KUKA KRL program: p01drop_newold.src, p01drop_newold.dat

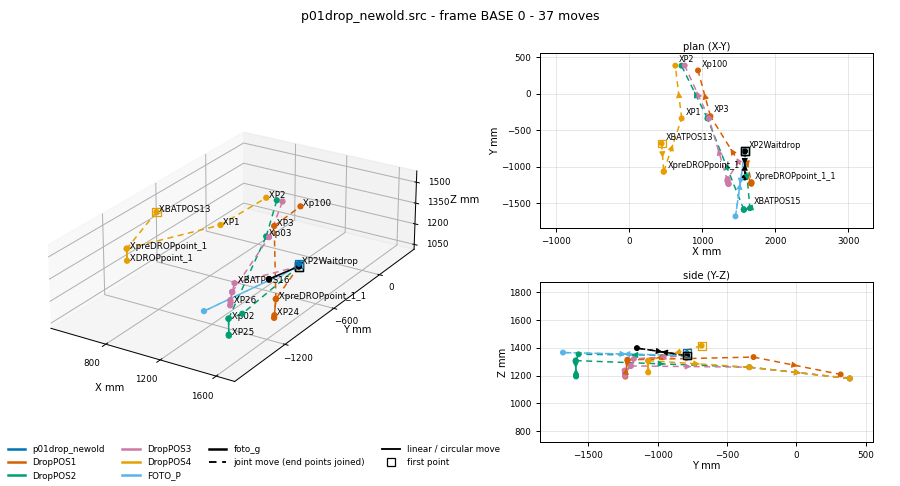
[picture p0: tool path of p01drop_newold.src in frame BASE 0, 37 of 40 moves have a stored position in this frame; points joined in program order, loops and branches not executed]
--- p01drop_newold.src ---
&ACCESS RVO1
&COMMENT Drop Part
&PARAM EDITMASK = *
&PARAM TEMPLATE = C:\KRC\Roboter\Template\vorgabe
&PARAM DISKPATH = KRC:\R1\Program\Sub Programs
DEF p01drop_newold( )
;FOLD INI
  ;FOLD BASISTECH INI

    GLOBAL INTERRUPT DECL 3 WHEN $STOPMESS==TRUE DO IR_STOPM ( )
    INTERRUPT ON 3
    BAS (#INITMOV,0 )
  ;ENDFOLD (BASISTECH INI)
;ENDFOLD (INI)
;================================================
; MODEL    : XXXX
; IE GROUP : XX
; STATION  : XXX
; ROBOT    : RX
; FUNCTION : Drop Part in StXX
;================================================
$TIMER[7]=0
$TIMER_STOP[7]=FALSE

waitarea:
QR_NOK=FALSE

;Wait For Area / Goto Safety / Return To Home
;FOLD PTP P2Waitdrop Vel=100 % PDAT2 Tool[8] Base[0];%{PE}%R 8.3.48,%MKUKATPBASIS,%CMOVE,%VPTP,%P 1:PTP, 2:P2Waitdrop, 3:, 5:100, 7:PDAT2
$BWDSTART=FALSE
PDAT_ACT=PPDAT2
FDAT_ACT=FP2Waitdrop
BAS(#PTP_PARAMS,100)
PTP XP2Waitdrop
;ENDFOLD

WAIT FOR ($IN[54]==TRUE) OR ($IN[1]==TRUE)

IF $in[54]==TRUE THEN
   bomberos_2 ( )               ; PICK In Station XX
ENDIF


;IF FALSE THEN

;Para de contar TC hasta que recibe typinfo para dejar (paleta indexada, tipo...)
$TIMER_STOP[7]=TRUE

;FOLD TYPE INFO

O_TYPE_REQ=FALSE
WAIT FOR I_TYPE_INFO==0
O_TYPE_REQ=TRUE
WAIT FOR ((I_TYPE_INFO>100) AND (I_TYPE_INFO<201) or ($IN[54]==TRUE))
IF $in[54]==TRUE THEN
   bomberos_2 ( )               ; PICK In Station XX
ENDIF
O_TYPE_INFO=I_TYPE_INFO

;ENDFOLD

;ENDIF

$TIMER_STOP[7]=FALSE

SWITCH i_TYPE_INFO ;coldplate grande o peq

CASE 111
$TIMER_STOP[7]=TRUE
INDICE_DROP=1

   O_TYPE_REQ=FALSE
;FOLD Fordtech.Area_Req Area Request: 3, Safety Position: 0, Return To Home: 0 ;%{PE}
Area_Req (3,0,0)
IF I_RETHP AND (0 <> 0) AND ($IN_HOME == TRUE) THEN
  GOTO PEXIT
ENDIF
;ENDFOLD
   $TIMER_STOP[7]=FALSE
   DropPOS1() ;POSICION 1 COLDPLATE GRANDE


CASE 112
$TIMER_STOP[7]=TRUE
INDICE_DROP=2

   O_TYPE_REQ=FALSE
;FOLD Fordtech.Area_Req Area Request: 3, Safety Position: 0, Return To Home: 0 ;%{PE}
Area_Req (3,0,0)
IF I_RETHP AND (0 <> 0) AND ($IN_HOME == TRUE) THEN
  GOTO PEXIT
ENDIF
;ENDFOLD
   $TIMER_STOP[7]=FALSE
   DropPOS2() ;POSICION 2 COLDPLATE GRANDE

CASE 113
$TIMER_STOP[7]=TRUE
INDICE_DROP=3

   O_TYPE_REQ=FALSE
;FOLD Fordtech.Area_Req Area Request: 3, Safety Position: 0, Return To Home: 0 ;%{PE}
Area_Req (3,0,0)
IF I_RETHP AND (0 <> 0) AND ($IN_HOME == TRUE) THEN
  GOTO PEXIT
ENDIF
;ENDFOLD
   $TIMER_STOP[7]=FALSE
   DropPOS3() ;POSICION 3 COLDPLATE GRANDE

CASE 150
bomberos_2 ()



CASE 121
$TIMER_STOP[7]=TRUE
INDICE_DROP=4

   O_TYPE_REQ=FALSE
;FOLD Fordtech.Area_Req Area Request: 3, Safety Position: 0, Return To Home: 0 ;%{PE}
Area_Req (3,0,0)
IF I_RETHP AND (0 <> 0) AND ($IN_HOME == TRUE) THEN
  GOTO PEXIT
ENDIF
;ENDFOLD
   $TIMER_STOP[7]=FALSE
   DropPOS1();POSICION 1 COLDPLATE PEQUEÑO

CASE 200
$TIMER_STOP[7]=TRUE
INDICE_DROP=4

   O_TYPE_REQ=FALSE
   P01DROP2_2();POSICION 1 COLDPLATE PEQUEÑO

DEFAULT

WAIT FOR FALSE

ENDSWITCH

;fold QR NOK
IF (QR_NOK==TRUE) THEN

GOTO waitarea
ENDIF

;ENDFOLD


;FOLD PROVISIONAL PARA PRUEBAS
IF M2_TYPE_INFO<13 THEN
M2_TYPE_INFO=M2_TYPE_INFO+1
ENDIF

;ENDFOLD

PEXIT:

;FOLD Guarda_TC Dejada

;Guarda TC dejada
$TIMER_STOP[7]=TRUE
TC_DROP[INDICE_DROP]=$TIMER[7]

IF (INDICE_DROP < 4) THEN ;CUANDO DEJA ARRAYS EN COLD PLATES GRANDES
   IF (INDICE_RACK == 1)THEN
      TC_CP_BIG[INDICE_DROP]=TC_DROP[INDICE_DROP]+TC_PICK_RACK1[INDICE_PICK]
   ELSE
      TC_CP_BIG[INDICE_DROP]=TC_DROP[INDICE_DROP]+TC_PICK_RACK2[INDICE_PICK]
   ENDIF
   IF (INDICE_DROP == 3) THEN ;Cuando rellena el tercer colplate acumula en array de CP big
      TC_ARRAY_CPB[INDICE_ARRAYS_CPB]=TC_CP_BIG[1]+TC_CP_BIG[2]+TC_CP_BIG[3]
      INDICE_ARRAYS_CPB=INDICE_ARRAYS_CPB+1
      IF (INDICE_ARRAYS_CPB > 18) THEN
         INDICE_ARRAYS_CPB=1
         ;Actualiza el tiempo de ciclo medio por bateria
         ;Toma el tiempo de ciclo medio por batería como la media de procesar 2 racks
         ;64 arrays y 4 cartones, eso vienen a ser unas 7 baterías y me sobra 1 array
         TC_MEDIO_CARTONES=((((TC_CARTON[1]+TC_CARTON[2]+TC_CARTON[3]+TC_CARTON[4])/1000)*63)/64)
         TC_MEDIO_BATERIA=((TC_ARRAY_CPB[1]+TC_ARRAY_CPB[2]+TC_ARRAY_CPB[3]+TC_ARRAY_CPB[4]+TC_ARRAY_CPB[5]+TC_ARRAY_CPB[6]+TC_ARRAY_CPB[7]+TC_ARRAY_CPB[8]+TC_ARRAY_CPB[9]+TC_ARRAY_CPB[10]+TC_ARRAY_CPB[11]+TC_ARRAY_CPB[12]+TC_ARRAY_CPB[13]+TC_ARRAY_CPB[14]+TC_ARRAY_CPB[15]+TC_ARRAY_CPB[16]+TC_ARRAY_CPB[17]+TC_ARRAY_CPB[18]+TC_CP_SMALL[1]+TC_CP_SMALL[2]+TC_CP_SMALL[3]+TC_CP_SMALL[4]+TC_CP_SMALL[5]+TC_CP_SMALL[6]+TC_CP_SMALL[7]+TC_CP_SMALL[8]+TC_CP_SMALL[9])/1000)
         TC_MEDIO_BATERIA=((TC_MEDIO_BATERIA+TC_MEDIO_CARTONES)/9)
      ENDIF
   ENDIF
      ENDIF

IF (INDICE_DROP == 4) THEN ;CUANDO DEJA ARRAYS EN COLD PLATE PEQUEÑOS
   IF (INDICE_RACK == 1)THEN
      TC_CP_SMALL[INDICE_ARRAYS_CPS]=TC_DROP[4]+TC_PICK_RACK1[INDICE_PICK]
   ELSE
      TC_CP_SMALL[INDICE_ARRAYS_CPS]=TC_DROP[4]+TC_PICK_RACK2[INDICE_PICK]
   ENDIF
   INDICE_ARRAYS_CPS=INDICE_ARRAYS_CPS+1
   IF (INDICE_ARRAYS_CPS > 9) THEN
      INDICE_ARRAYS_CPS=1
   ENDIF
ENDIF

;ENDFOLD

END
DEF       DropPOS1()



;FOLD PTP P11 CONT Vel=100 % PDAT29 Tool[8] Base[0];%{PE}%R 8.3.48,%MKUKATPBASIS,%CMOVE,%VPTP,%P 1:PTP, 2:P11, 3:C_DIS, 5:100, 7:PDAT29
$BWDSTART=FALSE
PDAT_ACT=PPDAT29
FDAT_ACT=FP11
BAS(#PTP_PARAMS,100)
PTP XP11 C_DIS
;ENDFOLD

;Wait For Area / Goto Safety / Return To Home

;FOLD PTP preDROPpoint_1_1 CONT Vel=100 % PDAT9 Tool[8] Base[0];%{PE}%R 8.3.48,%MKUKATPBASIS,%CMOVE,%VPTP,%P 1:PTP, 2:preDROPpoint_1_1, 3:C_DIS, 5:100, 7:PDAT9
$BWDSTART=FALSE
PDAT_ACT=PPDAT9
FDAT_ACT=FpreDROPpoint_1_1
BAS(#PTP_PARAMS,100)
PTP XpreDROPpoint_1_1 C_DIS
;ENDFOLD

;FOLD LIN P24 CONT Vel=2 m/s CPDAT10 Tool[8] Base[0];%{PE}%R 8.3.48,%MKUKATPBASIS,%CMOVE,%VLIN,%P 1:LIN, 2:P24, 3:C_DIS C_DIS, 5:2, 7:CPDAT10
$BWDSTART=FALSE
LDAT_ACT=LCPDAT10
FDAT_ACT=FP24
BAS(#CP_PARAMS,2)
LIN XP24 C_DIS C_DIS
;ENDFOLD
;FOLD LIN DROPpoint_1_1 Vel=0.02 m/s L Tool[8] Base[0];%{PE}%R 8.3.48,%MKUKATPBASIS,%CMOVE,%VLIN,%P 1:LIN, 2:DROPpoint_1_1, 3:, 5:0.02, 7:L
$BWDSTART=FALSE
LDAT_ACT=LL
FDAT_ACT=FDROPpoint_1_1
BAS(#CP_PARAMS,0.02)
LIN XDROPpoint_1_1
;ENDFOLD


;chequeo finales de carrera pieza ON
;FOLD WAIT FOR ( IN 257 'F carrera superior S202' );%{PE}%R 8.3.48,%MKUKATPBASIS,%CEXT_WAIT_FOR,%VEXT_WAIT_FOR,%P 2:, 4:, 5:$IN, 6:257, 7:F carrera superior S202, 9:
WAIT FOR  ( $IN[257] )
;ENDFOLD
;FOLD WAIT FOR ( IN 258 'F carrera superior S201' );%{PE}%R 8.3.48,%MKUKATPBASIS,%CEXT_WAIT_FOR,%VEXT_WAIT_FOR,%P 2:, 4:, 5:$IN, 6:258, 7:F carrera superior S201, 9:
WAIT FOR  ( $IN[258] )
;ENDFOLD

;abrir gara
cil_bat_reposo()

;chequeo sensores pieza OFF
;FOLD WAIT FOR NOT ( IN 243 'Partcheck array LH S501' );%{PE}%R 8.3.48,%MKUKATPBASIS,%CEXT_WAIT_FOR,%VEXT_WAIT_FOR,%P 2:NOT, 4:, 5:$IN, 6:243, 7:Partcheck array LH S501, 9:
WAIT FOR  NOT ( $IN[243] )
;ENDFOLD
;FOLD WAIT FOR NOT ( IN 244 'Partcheck array RH S502' );%{PE}%R 8.3.48,%MKUKATPBASIS,%CEXT_WAIT_FOR,%VEXT_WAIT_FOR,%P 2:NOT, 4:, 5:$IN, 6:244, 7:Partcheck array RH S502, 9:
WAIT FOR  NOT ( $IN[244] )
;ENDFOLD

;FOLD PTP preDROPpoint_1_1 CONT Vel=70 % PDAT20 Tool[8] Base[0];%{PE}%R 8.3.48,%MKUKATPBASIS,%CMOVE,%VPTP,%P 1:PTP, 2:preDROPpoint_1_1, 3:C_DIS, 5:70, 7:PDAT20
$BWDSTART=FALSE
PDAT_ACT=PPDAT20
FDAT_ACT=FpreDROPpoint_1_1
BAS(#PTP_PARAMS,70)
PTP XpreDROPpoint_1_1 C_DIS
;ENDFOLD

;chequeo finales de carrera pieza OFF
;FOLD WAIT FOR NOT ( IN 257 'F carrera superior S202' );%{PE}%R 8.3.48,%MKUKATPBASIS,%CEXT_WAIT_FOR,%VEXT_WAIT_FOR,%P 2:NOT, 4:, 5:$IN, 6:257, 7:F carrera superior S202, 9:
WAIT FOR  NOT ( $IN[257] )
;ENDFOLD
;FOLD WAIT FOR NOT ( IN 258 'F carrera superior S201' );%{PE}%R 8.3.48,%MKUKATPBASIS,%CEXT_WAIT_FOR,%VEXT_WAIT_FOR,%P 2:NOT, 4:, 5:$IN, 6:258, 7:F carrera superior S201, 9:
WAIT FOR  NOT ( $IN[258] )
;ENDFOLD

;FOLD SYN OUT 43 'Job Ready 3' State=TRUE at START Delay=0 ms;%{PE}%R 8.3.48,%MKUKATPBASIS,%COUT,%VSYNOUT,%P 2:43, 3:Job Ready 3, 5:TRUE, 7:0, 9:0, 12:0
TRIGGER WHEN DISTANCE=0 DELAY=0 DO $OUT[43]=TRUE
;ENDFOLD



;FOLD PTP P3 CONT Vel=100 % PDAT9 Tool[5] Base[0];%{PE}%R 8.3.48,%MKUKATPBASIS,%CMOVE,%VPTP,%P 1:PTP, 2:P3, 3:C_DIS, 5:100, 7:PDAT9
$BWDSTART=FALSE
PDAT_ACT=PPDAT9
FDAT_ACT=FP3
BAS(#PTP_PARAMS,100)
PTP XP3 C_DIS
;ENDFOLD

;Release Area 1
;FOLD SYN OUT 19 'Area Release 3' State=TRUE at START Delay=0 ms;%{PE}%R 8.3.48,%MKUKATPBASIS,%COUT,%VSYNOUT,%P 2:19, 3:Area Release 3, 5:TRUE, 7:0, 9:0, 12:0
TRIGGER WHEN DISTANCE=0 DELAY=0 DO $OUT[19]=TRUE
;ENDFOLD

;FOLD PTP p100 CONT Vel=100 % PDAT23 Tool[5] Base[0];%{PE}%R 8.3.48,%MKUKATPBASIS,%CMOVE,%VPTP,%P 1:PTP, 2:p100, 3:C_DIS, 5:100, 7:PDAT23
$BWDSTART=FALSE
PDAT_ACT=PPDAT23
FDAT_ACT=Fp100
BAS(#PTP_PARAMS,100)
PTP Xp100 C_DIS
;ENDFOLD


;FOLD PTP HOME Vel=100 % DEFAULT;%{PE}%R 8.3.48,%MKUKATPBASIS,%CMOVE,%VPTP,%P 1:PTP, 2:HOME, 3:, 5:100, 7:DEFAULT
$BWDSTART=FALSE
PDAT_ACT=PDEFAULT
FDAT_ACT=FHOME
BAS(#PTP_PARAMS,100)
$H_POS=XHOME
PTP XHOME
;ENDFOLD
;Jump Adress
PEXIT:



END

DEF       DropPOS2()


;FOLD PTP P12 CONT Vel=100 % PDAT30 Tool[8] Base[0];%{PE}%R 8.3.48,%MKUKATPBASIS,%CMOVE,%VPTP,%P 1:PTP, 2:P12, 3:C_DIS, 5:100, 7:PDAT30
$BWDSTART=FALSE
PDAT_ACT=PPDAT30
FDAT_ACT=FP12
BAS(#PTP_PARAMS,100)
PTP XP12 C_DIS
;ENDFOLD

;FOLD PTP BATPOS15 CONT Vel=100 % PDAT11 Tool[8] Base[0];%{PE}%R 8.3.48,%MKUKATPBASIS,%CMOVE,%VPTP,%P 1:PTP, 2:BATPOS15, 3:C_DIS, 5:100, 7:PDAT11
$BWDSTART=FALSE
PDAT_ACT=PPDAT11
FDAT_ACT=FBATPOS15
BAS(#PTP_PARAMS,100)
PTP XBATPOS15 C_DIS
;ENDFOLD
;Wait For Area / Goto Safety / Return To Home
;predrop pos
;FOLD PTP p02 CONT Vel=100 % PDAT12 Tool[8] Base[0];%{PE}%R 8.3.48,%MKUKATPBASIS,%CMOVE,%VPTP,%P 1:PTP, 2:p02, 3:C_DIS, 5:100, 7:PDAT12
$BWDSTART=FALSE
PDAT_ACT=PPDAT12
FDAT_ACT=Fp02
BAS(#PTP_PARAMS,100)
PTP Xp02 C_DIS
;ENDFOLD
;FOLD LIN P25 CONT Vel=2 m/s CPDAT11 Tool[8] Base[0];%{PE}%R 8.3.48,%MKUKATPBASIS,%CMOVE,%VLIN,%P 1:LIN, 2:P25, 3:C_DIS C_DIS, 5:2, 7:CPDAT11
$BWDSTART=FALSE
LDAT_ACT=LCPDAT11
FDAT_ACT=FP25
BAS(#CP_PARAMS,2)
LIN XP25 C_DIS C_DIS
;ENDFOLD
;drop pos
;FOLD LIN p01 Vel=0.02 m/s L Tool[8] Base[0];%{PE}%R 8.3.48,%MKUKATPBASIS,%CMOVE,%VLIN,%P 1:LIN, 2:p01, 3:, 5:0.02, 7:L
$BWDSTART=FALSE
LDAT_ACT=LL
FDAT_ACT=Fp01
BAS(#CP_PARAMS,0.02)
LIN Xp01
;ENDFOLD

;chequeo finales de carrera pieza ON
;FOLD WAIT FOR ( IN 257 'F carrera superior S202' );%{PE}%R 8.3.48,%MKUKATPBASIS,%CEXT_WAIT_FOR,%VEXT_WAIT_FOR,%P 2:, 4:, 5:$IN, 6:257, 7:F carrera superior S202, 9:
WAIT FOR  ( $IN[257] )
;ENDFOLD
;FOLD WAIT FOR ( IN 258 'F carrera superior S201' );%{PE}%R 8.3.48,%MKUKATPBASIS,%CEXT_WAIT_FOR,%VEXT_WAIT_FOR,%P 2:, 4:, 5:$IN, 6:258, 7:F carrera superior S201, 9:
WAIT FOR  ( $IN[258] )
;ENDFOLD

;abrir gara
cil_bat_reposo()

;chequeo sensores pieza OFF
;FOLD WAIT FOR NOT ( IN 243 'Partcheck array LH S501' );%{PE}%R 8.3.48,%MKUKATPBASIS,%CEXT_WAIT_FOR,%VEXT_WAIT_FOR,%P 2:NOT, 4:, 5:$IN, 6:243, 7:Partcheck array LH S501, 9:
WAIT FOR  NOT ( $IN[243] )
;ENDFOLD
;FOLD WAIT FOR NOT ( IN 244 'Partcheck array RH S502' );%{PE}%R 8.3.48,%MKUKATPBASIS,%CEXT_WAIT_FOR,%VEXT_WAIT_FOR,%P 2:NOT, 4:, 5:$IN, 6:244, 7:Partcheck array RH S502, 9:
WAIT FOR  NOT ( $IN[244] )
;ENDFOLD

;FOLD PTP p02 CONT Vel=70 % PDAT21 Tool[8] Base[0];%{PE}%R 8.3.48,%MKUKATPBASIS,%CMOVE,%VPTP,%P 1:PTP, 2:p02, 3:C_DIS, 5:70, 7:PDAT21
$BWDSTART=FALSE
PDAT_ACT=PPDAT21
FDAT_ACT=Fp02
BAS(#PTP_PARAMS,70)
PTP Xp02 C_DIS
;ENDFOLD


;chequeo finales de carrera pieza OFF
;FOLD WAIT FOR NOT ( IN 257 'F carrera superior S202' );%{PE}%R 8.3.48,%MKUKATPBASIS,%CEXT_WAIT_FOR,%VEXT_WAIT_FOR,%P 2:NOT, 4:, 5:$IN, 6:257, 7:F carrera superior S202, 9:
WAIT FOR  NOT ( $IN[257] )
;ENDFOLD
;FOLD WAIT FOR NOT ( IN 258 'F carrera superior S201' );%{PE}%R 8.3.48,%MKUKATPBASIS,%CEXT_WAIT_FOR,%VEXT_WAIT_FOR,%P 2:NOT, 4:, 5:$IN, 6:258, 7:F carrera superior S201, 9:
WAIT FOR  NOT ( $IN[258] )
;ENDFOLD

;FOLD SYN OUT 43 'Job Ready 3' State=TRUE at START Delay=0 ms;%{PE}%R 8.3.48,%MKUKATPBASIS,%COUT,%VSYNOUT,%P 2:43, 3:Job Ready 3, 5:TRUE, 7:0, 9:0, 12:0
TRIGGER WHEN DISTANCE=0 DELAY=0 DO $OUT[43]=TRUE
;ENDFOLD

;FOLD PTP p03 CONT Vel=100 % PDAT13 Tool[5] Base[0];%{PE}%R 8.3.48,%MKUKATPBASIS,%CMOVE,%VPTP,%P 1:PTP, 2:p03, 3:C_DIS, 5:100, 7:PDAT13
$BWDSTART=FALSE
PDAT_ACT=PPDAT13
FDAT_ACT=Fp03
BAS(#PTP_PARAMS,100)
PTP Xp03 C_DIS
;ENDFOLD

;Release Area 1
;FOLD SYN OUT 19 'Area Release 3' State=TRUE at START Delay=0 ms;%{PE}%R 8.3.48,%MKUKATPBASIS,%COUT,%VSYNOUT,%P 2:19, 3:Area Release 3, 5:TRUE, 7:0, 9:0, 12:0
TRIGGER WHEN DISTANCE=0 DELAY=0 DO $OUT[19]=TRUE
;ENDFOLD


;FOLD PTP p04 CONT Vel=100 % PDAT14 Tool[5] Base[0];%{PE}%R 8.3.48,%MKUKATPBASIS,%CMOVE,%VPTP,%P 1:PTP, 2:p04, 3:C_DIS, 5:100, 7:PDAT14
$BWDSTART=FALSE
PDAT_ACT=PPDAT14
FDAT_ACT=Fp04
BAS(#PTP_PARAMS,100)
PTP Xp04 C_DIS
;ENDFOLD

;FOLD PTP HOME Vel=100 % DEFAULT;%{PE}%R 8.3.48,%MKUKATPBASIS,%CMOVE,%VPTP,%P 1:PTP, 2:HOME, 3:, 5:100, 7:DEFAULT
$BWDSTART=FALSE
PDAT_ACT=PDEFAULT
FDAT_ACT=FHOME
BAS(#PTP_PARAMS,100)
$H_POS=XHOME
PTP XHOME
;ENDFOLD
;Jump Adress
PEXIT:

END
DEF       DropPOS3()


;FOLD PTP P13 CONT Vel=100 % PDAT31 Tool[8] Base[0];%{PE}%R 8.3.48,%MKUKATPBASIS,%CMOVE,%VPTP,%P 1:PTP, 2:P13, 3:C_DIS, 5:100, 7:PDAT31
$BWDSTART=FALSE
PDAT_ACT=PPDAT31
FDAT_ACT=FP13
BAS(#PTP_PARAMS,100)
PTP XP13 C_DIS
;ENDFOLD

;FOLD PTP BATPOS16 CONT Vel=100 % PDAT17 Tool[8] Base[0];%{PE}%R 8.3.48,%MKUKATPBASIS,%CMOVE,%VPTP,%P 1:PTP, 2:BATPOS16, 3:C_DIS, 5:100, 7:PDAT17
$BWDSTART=FALSE
PDAT_ACT=PPDAT17
FDAT_ACT=FBATPOS16
BAS(#PTP_PARAMS,100)
PTP XBATPOS16 C_DIS
;ENDFOLD
;Wait For Area / Goto Safety / Return To Home
;predroppos
;FOLD PTP p06 CONT Vel=100 % PDAT16 Tool[8] Base[0];%{PE}%R 8.3.48,%MKUKATPBASIS,%CMOVE,%VPTP,%P 1:PTP, 2:p06, 3:C_DIS, 5:100, 7:PDAT16
$BWDSTART=FALSE
PDAT_ACT=PPDAT16
FDAT_ACT=Fp06
BAS(#PTP_PARAMS,100)
PTP Xp06 C_DIS
;ENDFOLD
;FOLD LIN P26 CONT Vel=2 m/s CPDAT12 Tool[8] Base[0];%{PE}%R 8.3.48,%MKUKATPBASIS,%CMOVE,%VLIN,%P 1:LIN, 2:P26, 3:C_DIS C_DIS, 5:2, 7:CPDAT12
$BWDSTART=FALSE
LDAT_ACT=LCPDAT12
FDAT_ACT=FP26
BAS(#CP_PARAMS,2)
LIN XP26 C_DIS C_DIS
;ENDFOLD
;droppos
;FOLD LIN p05 Vel=0.02 m/s L Tool[8] Base[0];%{PE}%R 8.3.48,%MKUKATPBASIS,%CMOVE,%VLIN,%P 1:LIN, 2:p05, 3:, 5:0.02, 7:L
$BWDSTART=FALSE
LDAT_ACT=LL
FDAT_ACT=Fp05
BAS(#CP_PARAMS,0.02)
LIN Xp05
;ENDFOLD

;chequeo finales de carrera pieza ON
;FOLD WAIT FOR ( IN 257 'F carrera superior S202' );%{PE}%R 8.3.48,%MKUKATPBASIS,%CEXT_WAIT_FOR,%VEXT_WAIT_FOR,%P 2:, 4:, 5:$IN, 6:257, 7:F carrera superior S202, 9:
WAIT FOR  ( $IN[257] )
;ENDFOLD
;FOLD WAIT FOR ( IN 258 'F carrera superior S201' );%{PE}%R 8.3.48,%MKUKATPBASIS,%CEXT_WAIT_FOR,%VEXT_WAIT_FOR,%P 2:, 4:, 5:$IN, 6:258, 7:F carrera superior S201, 9:
WAIT FOR  ( $IN[258] )
;ENDFOLD

;abrir gara
cil_bat_reposo()

;chequeo sensores pieza OFF
;FOLD WAIT FOR NOT ( IN 243 'Partcheck array LH S501' );%{PE}%R 8.3.48,%MKUKATPBASIS,%CEXT_WAIT_FOR,%VEXT_WAIT_FOR,%P 2:NOT, 4:, 5:$IN, 6:243, 7:Partcheck array LH S501, 9:
WAIT FOR  NOT ( $IN[243] )
;ENDFOLD
;FOLD WAIT FOR NOT ( IN 244 'Partcheck array RH S502' );%{PE}%R 8.3.48,%MKUKATPBASIS,%CEXT_WAIT_FOR,%VEXT_WAIT_FOR,%P 2:NOT, 4:, 5:$IN, 6:244, 7:Partcheck array RH S502, 9:
WAIT FOR  NOT ( $IN[244] )
;ENDFOLD

;FOLD LIN P14 CONT Vel=2 m/s CPDAT9 Tool[5] Base[0];%{PE}%R 8.3.48,%MKUKATPBASIS,%CMOVE,%VLIN,%P 1:LIN, 2:P14, 3:C_DIS C_DIS, 5:2, 7:CPDAT9
$BWDSTART=FALSE
LDAT_ACT=LCPDAT9
FDAT_ACT=FP14
BAS(#CP_PARAMS,2)
LIN XP14 C_DIS C_DIS
;ENDFOLD
;FOLD PTP p06 CONT Vel=70 % PDAT22 Tool[8] Base[0];%{PE}%R 8.3.48,%MKUKATPBASIS,%CMOVE,%VPTP,%P 1:PTP, 2:p06, 3:C_DIS, 5:70, 7:PDAT22
$BWDSTART=FALSE
PDAT_ACT=PPDAT22
FDAT_ACT=Fp06
BAS(#PTP_PARAMS,70)
PTP Xp06 C_DIS
;ENDFOLD


;chequeo finales de carrera pieza OFF
;FOLD WAIT FOR NOT ( IN 257 'F carrera superior S202' );%{PE}%R 8.3.48,%MKUKATPBASIS,%CEXT_WAIT_FOR,%VEXT_WAIT_FOR,%P 2:NOT, 4:, 5:$IN, 6:257, 7:F carrera superior S202, 9:
WAIT FOR  NOT ( $IN[257] )
;ENDFOLD
;FOLD WAIT FOR NOT ( IN 258 'F carrera superior S201' );%{PE}%R 8.3.48,%MKUKATPBASIS,%CEXT_WAIT_FOR,%VEXT_WAIT_FOR,%P 2:NOT, 4:, 5:$IN, 6:258, 7:F carrera superior S201, 9:
WAIT FOR  NOT ( $IN[258] )
;ENDFOLD

;FOLD SYN OUT 43 'Job Ready 3' State=TRUE at START Delay=0 ms;%{PE}%R 8.3.48,%MKUKATPBASIS,%COUT,%VSYNOUT,%P 2:43, 3:Job Ready 3, 5:TRUE, 7:0, 9:0, 12:0
TRIGGER WHEN DISTANCE=0 DELAY=0 DO $OUT[43]=TRUE
;ENDFOLD

;FOLD PTP p07 CONT Vel=100 % PDAT18 Tool[5] Base[0];%{PE}%R 8.3.48,%MKUKATPBASIS,%CMOVE,%VPTP,%P 1:PTP, 2:p07, 3:C_DIS, 5:100, 7:PDAT18
$BWDSTART=FALSE
PDAT_ACT=PPDAT18
FDAT_ACT=Fp07
BAS(#PTP_PARAMS,100)
PTP Xp07 C_DIS
;ENDFOLD

;Release Area 1
;FOLD SYN OUT 19 'Area Release 3' State=TRUE at START Delay=0 ms;%{PE}%R 8.3.48,%MKUKATPBASIS,%COUT,%VSYNOUT,%P 2:19, 3:Area Release 3, 5:TRUE, 7:0, 9:0, 12:0
TRIGGER WHEN DISTANCE=0 DELAY=0 DO $OUT[19]=TRUE
;ENDFOLD


;FOLD PTP p08 CONT Vel=100 % PDAT19 Tool[5] Base[0];%{PE}%R 8.3.48,%MKUKATPBASIS,%CMOVE,%VPTP,%P 1:PTP, 2:p08, 3:C_DIS, 5:100, 7:PDAT19
$BWDSTART=FALSE
PDAT_ACT=PPDAT19
FDAT_ACT=Fp08
BAS(#PTP_PARAMS,100)
PTP Xp08 C_DIS
;ENDFOLD

;FOLD PTP HOME Vel=100 % DEFAULT;%{PE}%R 8.3.48,%MKUKATPBASIS,%CMOVE,%VPTP,%P 1:PTP, 2:HOME, 3:, 5:100, 7:DEFAULT
$BWDSTART=FALSE
PDAT_ACT=PDEFAULT
FDAT_ACT=FHOME
BAS(#PTP_PARAMS,100)
$H_POS=XHOME
PTP XHOME
;ENDFOLD
;Jump Adress
PEXIT:



END
DEF       DropPOS4()

;FOLD Fordtech.Area_Req Area Request: 3, Safety Position: 0, Return To Home: 0 ;%{PE}
Area_Req (3,0,0)
IF I_RETHP AND (0 <> 0) AND ($IN_HOME == TRUE) THEN
  GOTO PEXIT
ENDIF
;ENDFOLD

;FOLD PTP BATPOS13 Vel=100 % PDAT8 Tool[5] Base[0];%{PE}%R 8.3.48,%MKUKATPBASIS,%CMOVE,%VPTP,%P 1:PTP, 2:BATPOS13, 3:, 5:100, 7:PDAT8
$BWDSTART=FALSE
PDAT_ACT=PPDAT8
FDAT_ACT=FBATPOS13
BAS(#PTP_PARAMS,100)
PTP XBATPOS13
;ENDFOLD
;Wait For Area / Goto Safety / Return To Home

;FOLD PTP preDROPpoint_1 CONT Vel=100 % PDAT8 Tool[5] Base[0];%{PE}%R 8.3.48,%MKUKATPBASIS,%CMOVE,%VPTP,%P 1:PTP, 2:preDROPpoint_1, 3:C_DIS, 5:100, 7:PDAT8
$BWDSTART=FALSE
PDAT_ACT=PPDAT8
FDAT_ACT=FpreDROPpoint_1
BAS(#PTP_PARAMS,100)
PTP XpreDROPpoint_1 C_DIS
;ENDFOLD

;FOLD LIN DROPpoint_1 Vel=2 m/s CPDAT3 Tool[5] Base[0];%{PE}%R 8.3.48,%MKUKATPBASIS,%CMOVE,%VLIN,%P 1:LIN, 2:DROPpoint_1, 3:, 5:2, 7:CPDAT3
$BWDSTART=FALSE
LDAT_ACT=LCPDAT3
FDAT_ACT=FDROPpoint_1
BAS(#CP_PARAMS,2)
LIN XDROPpoint_1
;ENDFOLD

;abrir gara
cil_bat_reposo()

;FOLD LIN preDROPpoint_1 Vel=2 m/s CPDAT4 Tool[5] Base[0];%{PE}%R 8.3.48,%MKUKATPBASIS,%CMOVE,%VLIN,%P 1:LIN, 2:preDROPpoint_1, 3:, 5:2, 7:CPDAT4
$BWDSTART=FALSE
LDAT_ACT=LCPDAT4
FDAT_ACT=FpreDROPpoint_1
BAS(#CP_PARAMS,2)
LIN XpreDROPpoint_1
;ENDFOLD
;FOLD Fordtech.Job_Rdy Set Job Ready: 3   ;%{PE}
Job_Ready (3)
;ENDFOLD


;FOLD PTP P1 CONT Vel=100 % PDAT8 Tool[5] Base[0];%{PE}%R 8.3.48,%MKUKATPBASIS,%CMOVE,%VPTP,%P 1:PTP, 2:P1, 3:C_DIS, 5:100, 7:PDAT8
$BWDSTART=FALSE
PDAT_ACT=PPDAT8
FDAT_ACT=FP1
BAS(#PTP_PARAMS,100)
PTP XP1 C_DIS
;ENDFOLD
;FOLD PTP P2 CONT Vel=100 % PDAT8 Tool[5] Base[0];%{PE}%R 8.3.48,%MKUKATPBASIS,%CMOVE,%VPTP,%P 1:PTP, 2:P2, 3:C_DIS, 5:100, 7:PDAT8
$BWDSTART=FALSE
PDAT_ACT=PPDAT8
FDAT_ACT=FP2
BAS(#PTP_PARAMS,100)
PTP XP2 C_DIS
;ENDFOLD

;Release Area 1
;FOLD Fordtech.Area_Rel Area Release: 3   ;%{PE}
Area_Rel (3)
;ENDFOLD

;Jump Adress
PEXIT:




END

DEF      FOTO_P()


;FOLD PTP P17 CONT Vel=100 % PDAT34 Tool[5] Base[0];%{PE}%R 8.3.48,%MKUKATPBASIS,%CMOVE,%VPTP,%P 1:PTP, 2:P17, 3:C_DIS, 5:100, 7:PDAT34
$BWDSTART=FALSE
PDAT_ACT=PPDAT34
FDAT_ACT=FP17
BAS(#PTP_PARAMS,100)
PTP XP17 C_DIS
;ENDFOLD


;FOLD PTP P16 Vel=100 % PDAT33 Tool[5] Base[0];%{PE}%R 8.3.48,%MKUKATPBASIS,%CMOVE,%VPTP,%P 1:PTP, 2:P16, 3:, 5:100, 7:PDAT33
$BWDSTART=FALSE
PDAT_ACT=PPDAT33
FDAT_ACT=FP16
BAS(#PTP_PARAMS,100)
PTP XP16
;ENDFOLD

;FOLD OUT 953 'Reserve' State=TRUE CONT;%{PE}%R 8.3.48,%MKUKATPBASIS,%COUT,%VOUTX,%P 2:953, 3:Reserve, 5:TRUE, 6:CONTINUE
CONTINUE
$OUT[953]=TRUE
;ENDFOLD

;FOLD WAIT FOR ( IN 907 'Eines: Correccion X Bit 10' );%{PE}%R 8.3.48 %MKUKATPBASIS %CEXT_WAIT_FOR %VEXT_WAIT_FOR,%P 2:, 4:, 5:$IN, 6:907, 7:Eines: Correccion X Bit 10, 9:
WAIT FOR  ( $IN[907] )
;ENDFOLD

;FOLD OUT 953 'Reserve' State=FALSE CONT;%{PE}%R 8.3.48,%MKUKATPBASIS,%COUT,%VOUTX,%P 2:953, 3:Reserve, 5:FALSE, 6:CONTINUE
CONTINUE
$OUT[953]=FALSE
;ENDFOLD
;FOLD PTP P18 CONT Vel=100 % PDAT35 Tool[5] Base[0];%{PE}%R 8.3.48,%MKUKATPBASIS,%CMOVE,%VPTP,%P 1:PTP, 2:P18, 3:C_DIS, 5:100, 7:PDAT35
$BWDSTART=FALSE
PDAT_ACT=PPDAT35
FDAT_ACT=FP18
BAS(#PTP_PARAMS,100)
PTP XP18 C_DIS
;ENDFOLD
END

def      foto_g()


;FOLD PTP P19 CONT Vel=100 % PDAT36 Tool[5] Base[0];%{PE}%R 8.3.48,%MKUKATPBASIS,%CMOVE,%VPTP,%P 1:PTP, 2:P19, 3:C_DIS, 5:100, 7:PDAT36
$BWDSTART=FALSE
PDAT_ACT=PPDAT36
FDAT_ACT=FP19
BAS(#PTP_PARAMS,100)
PTP XP19 C_DIS
;ENDFOLD


;FOLD PTP P23 Vel=100 % PDAT39 Tool[5] Base[0];%{PE}%R 8.3.48,%MKUKATPBASIS,%CMOVE,%VPTP,%P 1:PTP, 2:P23, 3:, 5:100, 7:PDAT39
$BWDSTART=FALSE
PDAT_ACT=PPDAT39
FDAT_ACT=FP23
BAS(#PTP_PARAMS,100)
PTP XP23
;ENDFOLD

;FOLD OUT 953 'Reserve' State=TRUE CONT;%{PE}%R 8.3.48,%MKUKATPBASIS,%COUT,%VOUTX,%P 2:953, 3:Reserve, 5:TRUE, 6:CONTINUE
CONTINUE
$OUT[953]=TRUE
;ENDFOLD
;FOLD WAIT FOR ( IN 907 'Eines: Correccion X Bit 10' );%{PE}%R 8.3.48 %MKUKATPBASIS %CEXT_WAIT_FOR %VEXT_WAIT_FOR,%P 2:, 4:, 5:$IN, 6:907, 7:Eines: Correccion X Bit 10, 9:
WAIT FOR  ( $IN[907] )
;ENDFOLD


;FOLD OUT 953 'Reserve' State=FALSE CONT;%{PE}%R 8.3.48,%MKUKATPBASIS,%COUT,%VOUTX,%P 2:953, 3:Reserve, 5:FALSE, 6:CONTINUE
CONTINUE
$OUT[953]=FALSE
;ENDFOLD



;FOLD PTP P21 CONT Vel=100 % PDAT37 Tool[5] Base[0];%{PE}%R 8.3.48,%MKUKATPBASIS,%CMOVE,%VPTP,%P 1:PTP, 2:P21, 3:C_DIS, 5:100, 7:PDAT37
$BWDSTART=FALSE
PDAT_ACT=PPDAT37
FDAT_ACT=FP21
BAS(#PTP_PARAMS,100)
PTP XP21 C_DIS
;ENDFOLD

end

--- p01drop_newold.dat ---
&ACCESS RVO1
&COMMENT Drop Part
&PARAM EDITMASK = *
&PARAM TEMPLATE = C:\KRC\Roboter\Template\vorgabe
&PARAM DISKPATH = KRC:\R1\Program\Sub Programs
DEFDAT p01drop_newold

EXT  BAS (BAS_COMMAND  :IN,REAL  :IN )
DECL INT SUCCESS
;******************************
;*     E6POS Declarations     *
;******************************

DECL E6POS XP01WAITREQ2={X 2157.35596,Y -301.755188,Z 2852.14893,A -15.8183,B 72.8074417,C -9.82211304,S 2,T 34,E1 0.0,E2 0.0,E3 0.0,E4 0.0,E5 0.0,E6 0.0}
DECL E6POS XP10={X 2411.43896,Y 1748.73096,Z -1095.62903,A -177.692307,B -16.9195194,C 42.7874298,S 2,T 34,E1 0.0,E2 0.0,E3 0.0,E4 0.0,E5 0.0,E6 0.0}
DECL E6POS XP20={X 1670.59900,Y -157.831207,Z 2354.64209,A -15.8183,B 72.8074417,C -9.82211304,S 2,T 34,E1 0.0,E2 0.0,E3 0.0,E4 0.0,E5 0.0,E6 0.0}
DECL E6POS XP30={X 1670.59900,Y -157.831207,Z 2354.64209,A -15.8183,B 72.8074417,C -9.82211304,S 2,T 34,E1 0.0,E2 0.0,E3 0.0,E4 0.0,E5 0.0,E6 0.0}
DECL E6POS XDROP_POS={X 1670.59900,Y -157.831207,Z 2354.64209,A -15.8183,B 72.8074417,C -9.82211304,S 2,T 34,E1 0.0,E2 0.0,E3 0.0,E4 0.0,E5 0.0,E6 0.0}
DECL E6POS XP40={X 2411.43896,Y 1748.73096,Z -1095.62903,A -177.692307,B -16.9195194,C 42.7874298,S 2,T 34,E1 0.0,E2 0.0,E3 0.0,E4 0.0,E5 0.0,E6 0.0}
DECL E6POS XP50={X 2411.43896,Y 1748.73096,Z -1095.62903,A -177.692307,B -16.9195194,C 42.7874298,S 2,T 34,E1 0.0,E2 0.0,E3 0.0,E4 0.0,E5 0.0,E6 0.0}
DECL E6POS XP01WAITREL2={X 2411.43896,Y 1748.73096,Z -1095.62903,A -177.692307,B -16.9195194,C 42.7874298,S 2,T 34,E1 0.0,E2 0.0,E3 0.0,E4 0.0,E5 0.0,E6 0.0}

;******************************
;*     FDAT Declarations      *
;******************************

DECL FDAT FP01WAITREQ2={TOOL_NO 12,BASE_NO 0,IPO_FRAME #BASE}
DECL FDAT FP10={TOOL_NO 12,BASE_NO 0,IPO_FRAME #TCP}
DECL FDAT FP20={TOOL_NO 12,BASE_NO 0,IPO_FRAME #TCP}
DECL FDAT FP30={TOOL_NO 12,BASE_NO 0,IPO_FRAME #TCP}
DECL FDAT FDROP_POS={TOOL_NO 12,BASE_NO 0,IPO_FRAME #TCP}
DECL FDAT FP40={TOOL_NO 12,BASE_NO 0,IPO_FRAME #TCP}
DECL FDAT FP50={TOOL_NO 12,BASE_NO 0,IPO_FRAME #TCP}
DECL FDAT FP01WAITREL2={TOOL_NO 12,BASE_NO 0,IPO_FRAME #TCP}

;******************************
;*  PDAT & LDAT Declarations  *
;******************************

DECL PDAT PH={VEL 100.000,ACC 100.000,APO_DIST 100.000,APO_MODE #CDIS,GEAR_JERK 100.000,EXAX_IGN 0}

DECL MODULEPARAM_T LAST_TP_PARAMS={PARAMS[] "FORDTECH.P_AREA_REQ=3; FORDTECH.P_SAFETY_POS=0; FORDTECH.P_RET=0; Kuka.VelocityFieldEnabled=False; Kuka.ColDetectFieldEnabled=False; Kuka.MovementParameterFieldEnabled=False; Kuka.IsAngleEnabled=False; Kuka.PointName=P01Waitdrop; Kuka.FrameData.base_no=0; Kuka.FrameData.tool_no=12; Kuka.FrameData.ipo_frame=#BASE; Kuka.isglobalpoint=False; Kuka.MoveDataPtpName=H; Kuka.MovementDataPdat.apo_mode=#CDIS; Kuka.MovementDataPdat.apo_dist=100; Kuka.MovementData.vel=100; Kuka.MovementData.acc=100; Kuka.MovementData.exax_ign=0; Kuka.VelocityPtp=100; Kuka.BlendingEnabled=False; Kuka.APXEnabled=False; Kuka.CurrentCDSetIndex=0"}
DECL E6POS XP01Waitdrop={X 290.951508,Y 816.177185,Z 1155.55042,A -86.9976196,B 22.0779018,C -179.006119,S 6,T 27,E1 0.0,E2 0.0,E3 0.0,E4 0.0,E5 0.0,E6 0.0}
DECL FDAT FP01Waitdrop={TOOL_NO 5,BASE_NO 0,IPO_FRAME #BASE,POINT2[] " ",TQ_STATE FALSE}
DECL BASIS_SUGG_T LAST_BASIS={POINT1[] "P0                      ",POINT2[] "P0                      ",CP_PARAMS[] "CPDAT0                  ",PTP_PARAMS[] "PDAT0                   ",CONT[] "                        ",CP_VEL[] "0.02                    ",PTP_VEL[] "100                     ",SYNC_PARAMS[] "SYNCDAT                 ",SPL_NAME[] "S0                      ",A_PARAMS[] "ADAT0                   "}
DECL E6POS XP1WAITDROP={X -1019.53088,Y 1662.02295,Z 1494.18030,A -87.0150070,B 22.0766544,C -179.006226,S 6,T 27,E1 0.0,E2 0.0,E3 0.0,E4 0.0,E5 0.0,E6 0.0}
DECL FDAT FP1Waitdrop={TOOL_NO 12,BASE_NO 0,IPO_FRAME #BASE,POINT2[] " ",TQ_STATE FALSE}
DECL PDAT PPDAT1={VEL 100.000,ACC 100.000,APO_DIST 100.000,GEAR_JERK 50.0000,EXAX_IGN 0}
DECL E6POS XP2WAITDROP={X 1581.36292,Y -789.059875,Z 1362.23718,A 179.674332,B -0.834132493,C -179.411911,S 6,T 26,E1 0.0,E2 0.0,E3 0.0,E4 0.0,E5 0.0,E6 0.0}
DECL FDAT FP2Waitdrop={TOOL_NO 8,BASE_NO 0,IPO_FRAME #BASE,POINT2[] " ",TQ_STATE FALSE}
DECL PDAT PPDAT2={VEL 100.000,ACC 100.000,APO_DIST 100.000,GEAR_JERK 50.0000,EXAX_IGN 0}
DECL E6POS XP03drop_1={X 1357.71619,Y -332.386230,Z 1270.87256,A 92.5587387,B 7.42240524,C 175.886597,S 6,T 26,E1 0.0,E2 0.0,E3 0.0,E4 0.0,E5 0.0,E6 0.0}
DECL FDAT FP03drop_1={TOOL_NO 12,BASE_NO 0,IPO_FRAME #BASE,POINT2[] " ",TQ_STATE FALSE}
DECL PDAT PPDAT4={VEL 100.000,ACC 100.000,APO_DIST 100.000,GEAR_JERK 50.0000,EXAX_IGN 0}
DECL E6POS XP02drop_1={X 1435.38062,Y -451.789185,Z 1034.59302,A 89.9487686,B 4.10017967,C -172.489868,S 6,T 26,E1 0.0,E2 0.0,E3 0.0,E4 0.0,E5 0.0,E6 0.0}
DECL FDAT FP02drop_1={TOOL_NO 12,BASE_NO 0,IPO_FRAME #BASE,POINT2[] " ",TQ_STATE FALSE}
DECL PDAT PPDAT3={VEL 100.000,ACC 100.000,APO_DIST 100.000,GEAR_JERK 50.0000,EXAX_IGN 0}
DECL E6POS XP2={X 629.440857,Y 383.904541,Z 1179.93518,A -112.750427,B 20.1261520,C -170.604736,S 6,T 27,E1 0.0,E2 0.0,E3 0.0,E4 0.0,E5 0.0,E6 0.0}
DECL FDAT FP2={TOOL_NO 5,BASE_NO 0,IPO_FRAME #BASE,POINT2[] " ",TQ_STATE FALSE}
DECL PDAT PPDAT8={VEL 100.000,ACC 100.000,APO_DIST 100.000,APO_MODE #CDIS,GEAR_JERK 50.0000,EXAX_IGN 0}
DECL E6POS XP1={X 716.539490,Y -339.002350,Z 1261.05945,A -151.411957,B 9.54572201,C -170.760315,S 6,T 26,E1 0.0,E2 0.0,E3 0.0,E4 0.0,E5 0.0,E6 0.0}
DECL FDAT FP1={TOOL_NO 5,BASE_NO 0,IPO_FRAME #BASE,POINT2[] " ",TQ_STATE FALSE}
DECL PDAT PPDAT7={VEL 100.000,ACC 100.000,APO_DIST 100.000,APO_MODE #CDIS,GEAR_JERK 50.0000,EXAX_IGN 0}
DECL LDAT LCPDAT4={VEL 2.00000,ACC 100.000,APO_DIST 100.000,APO_FAC 50.0000,AXIS_VEL 100.000,AXIS_ACC 100.000,ORI_TYP #VAR,CIRC_TYP #BASE,JERK_FAC 50.0000,GEAR_JERK 50.0000,EXAX_IGN 0}
DECL E6POS XDROPpoint_1={X 471.147,Y -1067.04773,Z 1223.22400,A -179.451859,B -0.162765205,C 179.769058,S 6,T 26,E1 0.0,E2 0.0,E3 0.0,E4 0.0,E5 0.0,E6 0.0}
DECL FDAT FDROPpoint_1={TOOL_NO 5,BASE_NO 0,IPO_FRAME #BASE,POINT2[] " ",TQ_STATE FALSE}
DECL LDAT LCPDAT3={VEL 2.00000,ACC 100.000,APO_DIST 100.000,APO_FAC 50.0000,AXIS_VEL 100.000,AXIS_ACC 100.000,ORI_TYP #VAR,CIRC_TYP #BASE,JERK_FAC 50.0000,GEAR_JERK 50.0000,EXAX_IGN 0}
DECL E6POS XpreDROPpoint_1={X 471.147,Y -1067.04773,Z 1308.08960,A -179.451859,B -0.162765205,C 179.769058,S 6,T 26,E1 0.0,E2 0.0,E3 0.0,E4 0.0,E5 0.0,E6 0.0}
DECL FDAT FpreDROPpoint_1={TOOL_NO 5,BASE_NO 0,IPO_FRAME #BASE,POINT2[] " ",TQ_STATE FALSE}
DECL PDAT PPDAT6={VEL 100.000,ACC 100.000,APO_DIST 100.000,APO_MODE #CDIS,GEAR_JERK 50.0000,EXAX_IGN 0}
DECL E6POS XBATPOS13={X 442.124359,Y -682.465210,Z 1416.05603,A -171.206314,B 14.8656197,C -154.747955,S 6,T 26,E1 0.0,E2 0.0,E3 0.0,E4 0.0,E5 0.0,E6 0.0}
DECL FDAT FBATPOS13={TOOL_NO 5,BASE_NO 0,IPO_FRAME #BASE,POINT2[] " ",TQ_STATE FALSE}
DECL PDAT PPDAT5={VEL 100.000,ACC 100.000,APO_DIST 100.000,GEAR_JERK 50.0000,EXAX_IGN 0}
DECL E6POS XP4={X 197.117035,Y 1028.44482,Z 1209.08,A -97.8708878,B 5.08268261,C 175.164948,S 6,T 27,E1 0.0,E2 0.0,E3 0.0,E4 0.0,E5 0.0,E6 0.0}
DECL FDAT FP4={TOOL_NO 5,BASE_NO 0,IPO_FRAME #BASE,POINT2[] " ",TQ_STATE FALSE}
DECL E6POS XP3={X 1111.31909,Y -309.071167,Z 1333.85400,A 175.138336,B 11.3124800,C -177.333038,S 6,T 26,E1 0.0,E2 0.0,E3 0.0,E4 0.0,E5 0.0,E6 0.0}
DECL FDAT FP3={TOOL_NO 5,BASE_NO 0,IPO_FRAME #BASE,POINT2[] " ",TQ_STATE FALSE}
DECL LDAT LCPDAT6={VEL 2.00000,ACC 100.000,APO_DIST 100.000,APO_FAC 50.0000,AXIS_VEL 100.000,AXIS_ACC 100.000,ORI_TYP #VAR,CIRC_TYP #BASE,JERK_FAC 50.0000,GEAR_JERK 50.0000,EXAX_IGN 0}
DECL E6POS XDROPpoint_1_1={X 1670.14282,Y -1231.88098,Z 1193.25488,A 179.879410,B -0.278575361,C -179.995407,S 6,T 26,E1 0.0,E2 0.0,E3 0.0,E4 0.0,E5 0.0,E6 0.0}
DECL FDAT FDROPpoint_1_1={TOOL_NO 8,BASE_NO 0,IPO_FRAME #BASE,POINT2[] " ",TQ_STATE FALSE}
DECL LDAT LCPDAT5={VEL 2.00000,ACC 100.000,APO_DIST 100.000,APO_FAC 50.0000,AXIS_VEL 100.000,AXIS_ACC 100.000,ORI_TYP #VAR,CIRC_TYP #BASE,JERK_FAC 50.0000,GEAR_JERK 50.0000,EXAX_IGN 0}
DECL E6POS XpreDROPpoint_1_1={X 1672.14294,Y -1215.89258,Z 1314.19714,A 179.845,B -0.263878196,C -172.696686,S 6,T 26,E1 0.0,E2 0.0,E3 0.0,E4 0.0,E5 0.0,E6 0.0}
DECL FDAT FpreDROPpoint_1_1={TOOL_NO 8,BASE_NO 0,IPO_FRAME #BASE,POINT2[] " ",TQ_STATE FALSE}
DECL E6POS XBATPOS14={X 1672.14294,Y -789.059875,Z 1345.17505,A 179.845,B -0.263878196,C -172.696686,S 6,T 26,E1 0.0,E2 0.0,E3 0.0,E4 0.0,E5 0.0,E6 0.0}
DECL FDAT FBATPOS14={TOOL_NO 5,BASE_NO 0,IPO_FRAME #BASE,POINT2[] " ",TQ_STATE FALSE}
DECL PDAT PPDAT9={VEL 100.000,ACC 100.000,APO_DIST 100.000,APO_MODE #CDIS,GEAR_JERK 50.0000,EXAX_IGN 0}
DECL E6POS XP01={X 1568.78882,Y -1586.42542,Z 1194.44775,A -0.0518342331,B -0.113310046,C -179.391144,S 6,T 26,E1 0.0,E2 0.0,E3 0.0,E4 0.0,E5 0.0,E6 0.0}
DECL FDAT Fp01={TOOL_NO 8,BASE_NO 0,IPO_FRAME #BASE,POINT2[] " ",TQ_STATE FALSE}
DECL PDAT PPDAT10={VEL 100.000,ACC 100.000,APO_DIST 100.000,GEAR_JERK 50.0000,EXAX_IGN 0}
DECL LDAT LCPDAT1={VEL 2.00000,ACC 100.000,APO_DIST 100.000,APO_FAC 50.0000,AXIS_VEL 100.000,AXIS_ACC 100.000,ORI_TYP #VAR,CIRC_TYP #BASE,JERK_FAC 50.0000,GEAR_JERK 50.0000,EXAX_IGN 0}
DECL PDAT PPDAT11={VEL 100.000,ACC 100.000,APO_DIST 100.000,APO_MODE #CDIS,GEAR_JERK 50.0000,EXAX_IGN 0}
DECL E6POS XBATPOS15={X 1652.10083,Y -1568.82544,Z 1354.06287,A 12.7571592,B -2.70863843,C 176.134964,S 6,T 26,E1 0.0,E2 0.0,E3 0.0,E4 0.0,E5 0.0,E6 0.0}
DECL FDAT FBATPOS15={TOOL_NO 8,BASE_NO 0,IPO_FRAME #BASE,POINT2[] " ",TQ_STATE FALSE}
DECL E6POS XP02={X 1568.79468,Y -1589.39368,Z 1308.59436,A -0.0518342108,B -0.113310039,C -179.391144,S 6,T 26,E1 0.0,E2 0.0,E3 0.0,E4 0.0,E5 0.0,E6 0.0}
DECL FDAT Fp02={TOOL_NO 8,BASE_NO 0,IPO_FRAME #BASE,POINT2[] " ",TQ_STATE FALSE}
DECL PDAT PPDAT12={VEL 100.000,ACC 100.000,APO_DIST 100.000,APO_MODE #CDIS,GEAR_JERK 50.0000,EXAX_IGN 0}
DECL LDAT LCPDAT2={VEL 2.00000,ACC 100.000,APO_DIST 100.000,APO_FAC 50.0000,AXIS_VEL 100.000,AXIS_ACC 100.000,ORI_TYP #VAR,CIRC_TYP #BASE,JERK_FAC 50.0000,GEAR_JERK 50.0000,EXAX_IGN 0}
DECL PDAT PPDAT13={VEL 100.000,ACC 100.000,APO_DIST 100.000,APO_MODE #CDIS,GEAR_JERK 50.0000,EXAX_IGN 0}
DECL E6POS Xp03={X 1069.25427,Y -339.002350,Z 1261.05957,A -151.411957,B 9.54572392,C -170.760315,S 6,T 26,E1 0.0,E2 0.0,E3 0.0,E4 0.0,E5 0.0,E6 0.0}
DECL FDAT Fp03={TOOL_NO 5,BASE_NO 0,IPO_FRAME #BASE,POINT2[] " ",TQ_STATE FALSE}
DECL PDAT PPDAT14={VEL 100.000,ACC 100.000,APO_DIST 100.000,APO_MODE #CDIS,GEAR_JERK 50.0000,EXAX_IGN 0}
DECL E6POS Xp04={X 714.145325,Y 383.904541,Z 1179.93518,A -112.750427,B 20.1261520,C -170.604736,S 6,T 27,E1 0.0,E2 0.0,E3 0.0,E4 0.0,E5 0.0,E6 0.0}
DECL FDAT Fp04={TOOL_NO 5,BASE_NO 0,IPO_FRAME #BASE,POINT2[] " ",TQ_STATE FALSE}
DECL E6POS XP05={X 1356.28,Y -1234.52051,Z 1198.88123,A 179.687714,B -0.853233755,C 179.285538,S 6,T 26,E1 0.0,E2 0.0,E3 0.0,E4 0.0,E5 0.0,E6 0.0}
DECL FDAT Fp05={TOOL_NO 8,BASE_NO 0,IPO_FRAME #BASE,POINT2[] " ",TQ_STATE FALSE}
DECL PDAT PPDAT15={VEL 100.000,ACC 100.000,APO_DIST 100.000,APO_MODE #CDIS,GEAR_JERK 50.0000,EXAX_IGN 0}
DECL E6POS XP06={X 1344.35876,Y -1192.83325,Z 1270.12183,A -178.873672,B -2.07876205,C -178.198288,S 6,T 26,E1 0.0,E2 0.0,E3 0.0,E4 0.0,E5 0.0,E6 0.0}
DECL FDAT Fp06={TOOL_NO 8,BASE_NO 0,IPO_FRAME #BASE,POINT2[] " ",TQ_STATE FALSE}
DECL PDAT PPDAT16={VEL 100.000,ACC 100.000,APO_DIST 100.000,APO_MODE #CDIS,GEAR_JERK 50.0000,EXAX_IGN 0}
DECL PDAT PPDAT17={VEL 100.000,ACC 100.000,APO_DIST 100.000,APO_MODE #CDIS,GEAR_JERK 50.0000,EXAX_IGN 0}
DECL E6POS XBATPOS16={X 1347.29126,Y -1169.95642,Z 1321.72021,A -178.886719,B -2.07028890,C -178.139771,S 6,T 26,E1 0.0,E2 0.0,E3 0.0,E4 0.0,E5 0.0,E6 0.0}
DECL FDAT FBATPOS16={TOOL_NO 8,BASE_NO 0,IPO_FRAME #BASE,POINT2[] " ",TQ_STATE FALSE}
DECL LDAT LCPDAT7={VEL 2.00000,ACC 100.000,APO_DIST 100.000,APO_FAC 50.0000,AXIS_VEL 100.000,AXIS_ACC 100.000,ORI_TYP #VAR,CIRC_TYP #BASE,JERK_FAC 50.0000,GEAR_JERK 50.0000,EXAX_IGN 0}
DECL PDAT PPDAT18={VEL 100.000,ACC 100.000,APO_DIST 100.000,APO_MODE #CDIS,GEAR_JERK 50.0000,EXAX_IGN 0}
DECL E6POS Xp07={X 1090.57629,Y -339.002441,Z 1261.05957,A -151.411957,B 9.54572105,C -170.760315,S 6,T 26,E1 0.0,E2 0.0,E3 0.0,E4 0.0,E5 0.0,E6 0.0}
DECL FDAT Fp07={TOOL_NO 5,BASE_NO 0,IPO_FRAME #BASE,POINT2[] " ",TQ_STATE FALSE}
DECL PDAT PPDAT19={VEL 100.000,ACC 100.000,APO_DIST 100.000,APO_MODE #CDIS,GEAR_JERK 50.0000,EXAX_IGN 0}
DECL E6POS Xp08={X 758.473206,Y 385.849823,Z 1179.93518,A -112.750427,B 20.1261520,C -170.604736,S 6,T 27,E1 0.0,E2 0.0,E3 0.0,E4 0.0,E5 0.0,E6 0.0}
DECL FDAT Fp08={TOOL_NO 5,BASE_NO 0,IPO_FRAME #BASE,POINT2[] " ",TQ_STATE FALSE}
DECL LDAT LCPDAT8={VEL 2.00000,ACC 100.000,APO_DIST 100.000,APO_FAC 50.0000,AXIS_VEL 100.000,AXIS_ACC 100.000,ORI_TYP #VAR,CIRC_TYP #BASE,JERK_FAC 50.0000,GEAR_JERK 50.0000,EXAX_IGN 0}
DECL PDAT PPDAT20={VEL 100.000,ACC 100.000,APO_DIST 100.000,APO_MODE #CDIS,GEAR_JERK 50.0000,EXAX_IGN 0}
DECL PDAT PPDAT21={VEL 100.000,ACC 100.000,APO_DIST 100.000,APO_MODE #CDIS,GEAR_JERK 50.0000,EXAX_IGN 0}
DECL PDAT PPDAT22={VEL 100.000,ACC 100.000,APO_DIST 100.000,APO_MODE #CDIS,GEAR_JERK 50.0000,EXAX_IGN 0}
DECL E6POS XP100={X 940.903076,Y 318.277618,Z 1209.08,A -159.326324,B 5.08268261,C 175.164948,S 6,T 27,E1 0.0,E2 0.0,E3 0.0,E4 0.0,E5 0.0,E6 0.0}
DECL FDAT Fp100={TOOL_NO 5,BASE_NO 0,IPO_FRAME #BASE,POINT2[] " ",TQ_STATE FALSE}
DECL PDAT PPDAT23={VEL 100.000,ACC 100.000,APO_DIST 100.000,APO_MODE #CDIS,GEAR_JERK 50.0000,EXAX_IGN 0}
DECL E6POS XP5={X 1469.30664,Y -992.892761,Z 1336.18176,A 178.826553,B -0.278013229,C -177.836090,S 6,T 26,E1 0.0,E2 0.0,E3 0.0,E4 0.0,E5 0.0,E6 0.0}
DECL FDAT FP5={TOOL_NO 5,BASE_NO 0,IPO_FRAME #BASE,POINT2[] " ",TQ_STATE FALSE}
DECL PDAT PPDAT24={VEL 100.000,ACC 100.000,APO_DIST 100.000,APO_MODE #CDIS,GEAR_JERK 50.0000,EXAX_IGN 0}
DECL E6POS XP6={X 1481.10022,Y -1068.82,Z 1369.03247,A 179.760498,B -0.276004165,C -179.419418,S 6,T 26,E1 0.0,E2 0.0,E3 0.0,E4 0.0,E5 0.0,E6 0.0}
DECL FDAT FP6={TOOL_NO 5,BASE_NO 0,IPO_FRAME #BASE,POINT2[] " ",TQ_STATE FALSE}
DECL PDAT PPDAT25={VEL 100.000,ACC 100.000,APO_DIST 100.000,APO_MODE #CDIS,GEAR_JERK 50.0000,EXAX_IGN 0}
DECL E6POS XP7={X -467.506348,Y 1381.33057,Z 1221.24878,A -88.9552,B 22.2455826,C 175.857315,S 6,T 27,E1 0.0,E2 0.0,E3 0.0,E4 0.0,E5 0.0,E6 0.0}
DECL FDAT FP7={TOOL_NO 5,BASE_NO 0,IPO_FRAME #BASE,POINT2[] " ",TQ_STATE FALSE}
DECL PDAT PPDAT26={VEL 100.000,ACC 100.000,APO_DIST 100.000,APO_MODE #CDIS,GEAR_JERK 50.0000,EXAX_IGN 0}
DECL E6POS XP8={X -467.506348,Y 1381.33057,Z 1221.24878,A -88.9552,B 22.2455826,C 175.857315,S 6,T 27,E1 0.0,E2 0.0,E3 0.0,E4 0.0,E5 0.0,E6 0.0}
DECL FDAT FP8={TOOL_NO 5,BASE_NO 0,IPO_FRAME #BASE,POINT2[] " ",TQ_STATE FALSE}
DECL PDAT PPDAT27={VEL 100.000,ACC 100.000,APO_DIST 100.000,APO_MODE #CDIS,GEAR_JERK 50.0000,EXAX_IGN 0}
DECL E6POS XP9={X -467.506348,Y 1381.33057,Z 1221.24878,A -88.9552,B 22.2455826,C 175.857315,S 6,T 27,E1 0.0,E2 0.0,E3 0.0,E4 0.0,E5 0.0,E6 0.0}
DECL FDAT FP9={TOOL_NO 5,BASE_NO 0,IPO_FRAME #BASE,POINT2[] " ",TQ_STATE FALSE}
DECL PDAT PPDAT28={VEL 100.000,ACC 100.000,APO_DIST 100.000,APO_MODE #CDIS,GEAR_JERK 50.0000,EXAX_IGN 0}
DECL E6POS XP11={X 1581.36292,Y -789.059875,Z 1345.17505,A 179.845,B -0.263878018,C -172.696686,S 6,T 26,E1 0.0,E2 0.0,E3 0.0,E4 0.0,E5 0.0,E6 0.0}
DECL FDAT FP11={TOOL_NO 8,BASE_NO 0,IPO_FRAME #BASE,POINT2[] " ",TQ_STATE FALSE}
DECL PDAT PPDAT29={VEL 100.000,ACC 100.000,APO_DIST 100.000,APO_MODE #CDIS,GEAR_JERK 50.0000,EXAX_IGN 0}
DECL E6POS XP12={X 1581.36292,Y -789.059875,Z 1345.17505,A 179.845,B -0.263878018,C -172.696686,S 6,T 26,E1 0.0,E2 0.0,E3 0.0,E4 0.0,E5 0.0,E6 0.0}
DECL FDAT FP12={TOOL_NO 8,BASE_NO 0,IPO_FRAME #BASE,POINT2[] " ",TQ_STATE FALSE}
DECL PDAT PPDAT30={VEL 100.000,ACC 100.000,APO_DIST 100.000,APO_MODE #CDIS,GEAR_JERK 50.0000,EXAX_IGN 0}
DECL E6POS XP13={X 1581.36292,Y -789.059875,Z 1345.17505,A 179.845,B -0.263878018,C -172.696686,S 6,T 26,E1 0.0,E2 0.0,E3 0.0,E4 0.0,E5 0.0,E6 0.0}
DECL FDAT FP13={TOOL_NO 8,BASE_NO 0,IPO_FRAME #BASE,POINT2[] " ",TQ_STATE FALSE}
DECL PDAT PPDAT31={VEL 100.000,ACC 100.000,APO_DIST 100.000,APO_MODE #CDIS,GEAR_JERK 50.0000,EXAX_IGN 0}
DECL E6POS XP14={X 1359.54651,Y -1237.52588,Z 1237.19409,A 179.687714,B -0.853233755,C 179.285538,S 6,T 26,E1 0.0,E2 0.0,E3 0.0,E4 0.0,E5 0.0,E6 0.0}
DECL FDAT FP14={TOOL_NO 5,BASE_NO 0,IPO_FRAME #BASE,POINT2[] " ",TQ_STATE FALSE}
DECL LDAT LCPDAT9={VEL 2.00000,ACC 100.000,APO_DIST 100.000,APO_FAC 50.0000,AXIS_VEL 100.000,AXIS_ACC 100.000,ORI_TYP #VAR,CIRC_TYP #BASE,JERK_FAC 50.0000,GEAR_JERK 50.0000,EXAX_IGN 0}
DECL E6POS XP15={X 1581.36292,Y -789.059875,Z 1345.17505,A 179.845,B -0.263878196,C -172.696686,S 6,T 26,E1 0.0,E2 0.0,E3 0.0,E4 0.0,E5 0.0,E6 0.0}
DECL FDAT FP15={TOOL_NO 5,BASE_NO 0,IPO_FRAME #BASE,POINT2[] " ",TQ_STATE FALSE}
DECL PDAT PPDAT32={VEL 100.000,ACC 100.000,APO_DIST 100.000,GEAR_JERK 50.0000,EXAX_IGN 0}
DECL E6POS XP16={X 1454.24036,Y -1680.92651,Z 1366.54358,A -5.35814667,B -7.88578033,C 178.642899,S 6,T 26,E1 0.0,E2 0.0,E3 0.0,E4 0.0,E5 0.0,E6 0.0}
DECL FDAT FP16={TOOL_NO 5,BASE_NO 0,IPO_FRAME #BASE,POINT2[] " ",TQ_STATE FALSE}
DECL PDAT PPDAT33={VEL 100.000,ACC 100.000,APO_DIST 100.000,GEAR_JERK 50.0000,EXAX_IGN 0}
DECL E6POS XP17={X 1581.36292,Y -789.059875,Z 1345.17505,A 179.845,B -0.263878196,C -172.696686,S 6,T 26,E1 0.0,E2 0.0,E3 0.0,E4 0.0,E5 0.0,E6 0.0}
DECL FDAT FP17={TOOL_NO 5,BASE_NO 0,IPO_FRAME #BASE,POINT2[] " ",TQ_STATE FALSE}
DECL PDAT PPDAT34={VEL 100.000,ACC 100.000,APO_DIST 100.000,APO_MODE #CDIS,GEAR_JERK 50.0000,EXAX_IGN 0}
DECL E6POS XP18={X 1581.36292,Y -789.059875,Z 1345.17505,A 179.845,B -0.263878196,C -172.696686,S 6,T 26,E1 0.0,E2 0.0,E3 0.0,E4 0.0,E5 0.0,E6 0.0}
DECL FDAT FP18={TOOL_NO 5,BASE_NO 0,IPO_FRAME #BASE,POINT2[] " ",TQ_STATE FALSE}
DECL PDAT PPDAT35={VEL 100.000,ACC 100.000,APO_DIST 100.000,APO_MODE #CDIS,GEAR_JERK 50.0000,EXAX_IGN 0}
DECL E6POS XP19={X 1581.36292,Y -789.059875,Z 1345.17505,A 179.845,B -0.263878196,C -172.696686,S 6,T 26,E1 0.0,E2 0.0,E3 0.0,E4 0.0,E5 0.0,E6 0.0}
DECL FDAT FP19={TOOL_NO 5,BASE_NO 0,IPO_FRAME #BASE,POINT2[] " ",TQ_STATE FALSE}
DECL PDAT PPDAT36={VEL 100.000,ACC 100.000,APO_DIST 100.000,APO_MODE #CDIS,GEAR_JERK 50.0000,EXAX_IGN 0}
DECL E6POS XP21={X 1581.36292,Y -789.059875,Z 1345.17505,A 179.845,B -0.263878196,C -172.696686,S 6,T 26,E1 0.0,E2 0.0,E3 0.0,E4 0.0,E5 0.0,E6 0.0}
DECL FDAT FP21={TOOL_NO 5,BASE_NO 0,IPO_FRAME #BASE,POINT2[] " ",TQ_STATE FALSE}
DECL PDAT PPDAT37={VEL 100.000,ACC 100.000,APO_DIST 100.000,APO_MODE #CDIS,GEAR_JERK 50.0000,EXAX_IGN 0}
DECL E6POS XP22={X 1581.36292,Y -1115.88245,Z 1345.17505,A 179.845,B -0.263878196,C -172.696686,S 6,T 26,E1 0.0,E2 0.0,E3 0.0,E4 0.0,E5 0.0,E6 0.0}
DECL FDAT FP22={TOOL_NO 5,BASE_NO 0,IPO_FRAME #BASE,POINT2[] " ",TQ_STATE FALSE}
DECL PDAT PPDAT38={VEL 100.000,ACC 100.000,APO_DIST 100.000,GEAR_JERK 50.0000,EXAX_IGN 0}
DECL E6POS XP23={X 1581.36292,Y -1148.35986,Z 1398.59546,A 179.815231,B -0.243960768,C -165.986893,S 6,T 26,E1 0.0,E2 0.0,E3 0.0,E4 0.0,E5 0.0,E6 0.0}
DECL FDAT FP23={TOOL_NO 5,BASE_NO 0,IPO_FRAME #BASE,POINT2[] " ",TQ_STATE FALSE}
DECL PDAT PPDAT39={VEL 100.000,ACC 100.000,APO_DIST 100.000,GEAR_JERK 50.0000,EXAX_IGN 0}
DECL E6POS XP24={X 1672.14282,Y -1231.88513,Z 1211.24512,A 179.879410,B -0.278575361,C -179.995407,S 6,T 26,E1 0.0,E2 0.0,E3 0.0,E4 0.0,E5 0.0,E6 0.0}
DECL FDAT FP24={TOOL_NO 8,BASE_NO 0,IPO_FRAME #BASE,POINT2[] " ",TQ_STATE FALSE}
DECL LDAT LCPDAT10={VEL 2.00000,ACC 100.000,APO_DIST 100.000,APO_FAC 50.0000,AXIS_VEL 100.000,AXIS_ACC 100.000,ORI_TYP #VAR,CIRC_TYP #BASE,JERK_FAC 50.0000,GEAR_JERK 50.0000,EXAX_IGN 0}
DECL E6POS XP25={X 1567.79663,Y -1586.38220,Z 1200.89868,A -0.0518342145,B -0.113310039,C -179.391144,S 6,T 26,E1 0.0,E2 0.0,E3 0.0,E4 0.0,E5 0.0,E6 0.0}
DECL FDAT FP25={TOOL_NO 8,BASE_NO 0,IPO_FRAME #BASE,POINT2[] " ",TQ_STATE FALSE}
DECL LDAT LCPDAT11={VEL 2.00000,ACC 100.000,APO_DIST 100.000,APO_FAC 50.0000,AXIS_VEL 100.000,AXIS_ACC 100.000,ORI_TYP #VAR,CIRC_TYP #BASE,JERK_FAC 50.0000,GEAR_JERK 50.0000,EXAX_IGN 0}
DECL E6POS XP26={X 1359.71521,Y -1234.66870,Z 1217.57349,A 179.687714,B -0.853233755,C 179.285538,S 6,T 26,E1 0.0,E2 0.0,E3 0.0,E4 0.0,E5 0.0,E6 0.0}
DECL FDAT FP26={TOOL_NO 8,BASE_NO 0,IPO_FRAME #BASE,POINT2[] " ",TQ_STATE FALSE}
DECL LDAT LCPDAT12={VEL 2.00000,ACC 100.000,APO_DIST 100.000,APO_FAC 50.0000,AXIS_VEL 100.000,AXIS_ACC 100.000,ORI_TYP #VAR,CIRC_TYP #BASE,JERK_FAC 50.0000,GEAR_JERK 50.0000,EXAX_IGN 0}
DECL LDAT LL={VEL 2.00000,ACC 25.0000,APO_DIST 100.000,APO_FAC 50.0000,AXIS_VEL 100.000,AXIS_ACC 100.000,ORI_TYP #VAR,CIRC_TYP #BASE,JERK_FAC 50.0000,GEAR_JERK 50.0000,EXAX_IGN 0}
ENDDAT
